PROGRAM INPUT_G6
VAR
	TMR11: TON;
	TMR12: TON;
	TMR10: TON;
	TMR8: TON;
	TMR9: TON;
	TMR7: TON;
	TMR3: TON;
	TP1: TP;
	TMR1: TON;
	START_ROBOT: TP;
	TP2: TP;
	O_G6_HANG: BOOL;
	I_G6_HANG: BOOL;
	TMR2: TON;
	GO_ROBOT: BOOL;
	TP3: TP;
	TMR4: TON;
	CNT_CYCLE: CTU;
	START_ROTATE: R_TRIG;
	IN: INT;
	TP_END_FUKUDA: TP;
	CNT_END_FUKUDA: CTU;
	ROBOT_READY: BOOL;
	ROBOT_G6_READY: BOOL;
	END_FUKUDA: BOOL;
	O_END_FUKUDA: BOOL;
	TEMP_COUNTER_FUKUDA_A: INT;
	TEMP_COUNTER_FUKUDA_B: INT;
	O_END_FUKUDB: BOOL;
	MAX_DEVICE: INT;
	TMR_HANG: TON;
	GRP1: Tp;
	GRP2: Tp;
	GRP3: Tp;
	GRP4: Tp;
	CNT_PLACING: ctu;
	CNT_TAKING: CTU;
	CNT_CYCLE1: CTU;
END_VAR

VAR PERSISTENT
	TRGEN: R_TRIG;
END_VAR

IF INPUT_G6_VAR.I_G6_ENABLE  THEN
//GRIPPING 
IF INPUT_G6_VAR.IX_G6_GRIPPER_1 THEN
	INPUT_G6_VAR.O_G6_GRIPPER_CLOSE_1:=TRUE;
	INPUT_G6_VAR.O_G6_GRIPPER_OPEN_1:=FALSE;
ELSE
	INPUT_G6_VAR.O_G6_GRIPPER_CLOSE_1:=FALSE;
	INPUT_G6_VAR.O_G6_GRIPPER_OPEN_1:=TRUE;
END_IF

IF INPUT_G6_VAR.IX_G6_GRIPPER_2 THEN
	INPUT_G6_VAR.O_G6_GRIPPER_CLOSE_2:=TRUE;
	INPUT_G6_VAR.O_G6_GRIPPER_OPEN_2:=FALSE;
ELSE
	INPUT_G6_VAR.O_G6_GRIPPER_CLOSE_2:=FALSE;
	INPUT_G6_VAR.O_G6_GRIPPER_OPEN_2:=TRUE;
END_IF 

IF INPUT_G6_VAR.IX_G6_GRIPPER_3 THEN
	INPUT_G6_VAR.O_G6_GRIPPER_CLOSE_3:=TRUE;
	INPUT_G6_VAR.O_G6_GRIPPER_OPEN_3:=FALSE;
ELSE
	INPUT_G6_VAR.O_G6_GRIPPER_CLOSE_3:=FALSE;
	INPUT_G6_VAR.O_G6_GRIPPER_OPEN_3:=TRUE;
END_IF

IF INPUT_G6_VAR.IX_G6_GRIPPER_4 THEN
	INPUT_G6_VAR.O_G6_GRIPPER_CLOSE_4:=TRUE;
	INPUT_G6_VAR.O_G6_GRIPPER_OPEN_4:=FALSE;
ELSE
	INPUT_G6_VAR.O_G6_GRIPPER_CLOSE_4:=FALSE;
	INPUT_G6_VAR.O_G6_GRIPPER_OPEN_4:=TRUE;
END_IF

//EXTENDER DOWN
IF INPUT_G6_VAR.IX_G6_GRIPPER_EXT_1 THEN
	INPUT_G6_VAR.O_G6_GRIPPER_EXT_DOWN_1:=TRUE;
	INPUT_G6_VAR.O_G6_GRIPPER_EXT_UP_1:=FALSE;
ELSE
	INPUT_G6_VAR.O_G6_GRIPPER_EXT_DOWN_1:=FALSE;
	INPUT_G6_VAR.O_G6_GRIPPER_EXT_UP_1:=TRUE;
END_IF

IF INPUT_G6_VAR.IX_G6_GRIPPER_EXT_2 THEN
	INPUT_G6_VAR.O_G6_GRIPPER_EXT_DOWN_2:=TRUE;
	INPUT_G6_VAR.O_G6_GRIPPER_EXT_UP_2:=FALSE;
ELSE
	INPUT_G6_VAR.O_G6_GRIPPER_EXT_DOWN_2:=FALSE;
	INPUT_G6_VAR.O_G6_GRIPPER_EXT_UP_2:=TRUE;
END_IF

IF INPUT_G6_VAR.IX_G6_GRIPPER_EXT_3 THEN
	INPUT_G6_VAR.O_G6_GRIPPER_EXT_DOWN_3:=TRUE;
	INPUT_G6_VAR.O_G6_GRIPPER_EXT_UP_3:=FALSE;
ELSE
	INPUT_G6_VAR.O_G6_GRIPPER_EXT_DOWN_3:=FALSE;
	INPUT_G6_VAR.O_G6_GRIPPER_EXT_UP_3:=TRUE;
END_IF

IF INPUT_G6_VAR.IX_G6_GRIPPER_EXT_4 THEN
	INPUT_G6_VAR.O_G6_GRIPPER_EXT_DOWN_4:=TRUE;
	INPUT_G6_VAR.O_G6_GRIPPER_EXT_UP_4:=FALSE;
ELSE
	INPUT_G6_VAR.O_G6_GRIPPER_EXT_DOWN_4:=FALSE;
	INPUT_G6_VAR.O_G6_GRIPPER_EXT_UP_4:=TRUE;
END_IF
IF INPUT_G6_VAR.I_G6_READY_TAKEUP THEN
	INPUT_G6_VAR.O_G6_GRIPPER_CLOSE_1:=FALSE;
	INPUT_G6_VAR.O_G6_GRIPPER_OPEN_1:=TRUE;
	
	INPUT_G6_VAR.O_G6_GRIPPER_CLOSE_2:=FALSE;
	INPUT_G6_VAR.O_G6_GRIPPER_OPEN_2:=TRUE;
	
	INPUT_G6_VAR.O_G6_GRIPPER_CLOSE_3:=FALSE;
	INPUT_G6_VAR.O_G6_GRIPPER_OPEN_3:=TRUE;
	
	INPUT_G6_VAR.O_G6_GRIPPER_CLOSE_3:=FALSE;
	INPUT_G6_VAR.O_G6_GRIPPER_OPEN_3:=TRUE;
END_IF

INPUT_G6_VAR.GRIPPER_OPEN_1:=INPUT_G6_VAR.I_G6_GRIPPER_OPEN_1;
INPUT_G6_VAR.GRIPPER_OPEN_2:=INPUT_G6_VAR.I_G6_GRIPPER_OPEN_2;
INPUT_G6_VAR.GRIPPER_OPEN_3:=INPUT_G6_VAR.I_G6_GRIPPER_OPEN_3;
INPUT_G6_VAR.GRIPPER_OPEN_4:=INPUT_G6_VAR.I_G6_GRIPPER_OPEN_4;

INPUT_G6_VAR.GRIPPER_CLOSE_1:=INPUT_G6_VAR.I_G6_GRIPPER_CLOSE_1;
INPUT_G6_VAR.GRIPPER_CLOSE_2:=INPUT_G6_VAR.I_G6_GRIPPER_CLOSE_2;
INPUT_G6_VAR.GRIPPER_CLOSE_3:=INPUT_G6_VAR.I_G6_GRIPPER_CLOSE_3;
INPUT_G6_VAR.GRIPPER_CLOSE_4:=INPUT_G6_VAR.I_G6_GRIPPER_CLOSE_4;

//ACTIVATE ROBOT
TRGEN(CLK:=INPUT_G6_VAR.I_G6_ENABLE); 
IF TRGEN.Q THEN
	INPUT_G6_VAR.O_G6_RESET_COUNTER_PICK:=TRUE;
END_IF
IF INPUT_G6_VAR.I_G6_START_PLACING OR INPUT_G6_VAR.I_G6_START_TAKEUP THEN
	INPUT_G6_VAR.O_G6_RESET_COUNTER_PICK:=FALSE;
END_IF
//IF INPUT_G6_VAR.I_G6_ENABLE THEN
TP_END_FUKUDA(IN:=INPUT_G6_VAR.I_G6_END_FUKUDA,PT:=T#0.1S);
CNT_END_FUKUDA(CU:=TP_END_FUKUDA.Q,RESET:=CNT_END_FUKUDA.Q,PV:=1000);

INPUT_VAR.I_STOPPER_TRANSFER_ON_A:= INPUT_VAR.O_STOPPER_TRANSFER_A;
//IF INPUT_VAR.I_STOPPER_TRANSFER_ON_A OR INPUT_VAR.I_STOPPER_TRANSFER_ON_B THEN
INPUT_G6_VAR.O_G6_SETMOTOROFF:=FALSE;
IF NOT INPUT_G6_VAR.I_G6_MOTORON THEN
	INPUT_G6_VAR.O_G6_STOP:=FALSE;
END_IF
IF NOT INPUT_G6_VAR.I_G6_MOTORON AND INPUT_G6_VAR.I_G6_READY AND NOT INPUT_G6_VAR.I_G6_ESTOPON AND NOT INPUT_G6_VAR.I_G6_SAFEGUARDON THEN
	INPUT_G6_VAR.O_G6_SETMOTORON:=TRUE;
	INPUT_G6_VAR.O_G6_STOP:=FALSE;
	INPUT_G6_VAR.O_G6_RESET :=FALSE;	
	INPUT_G6_VAR.O_G6_START :=FALSE ;
	INPUT_G6_VAR.O_G6_CONTINUE :=FALSE;
TMR1(IN:=INPUT_G6_VAR.O_G6_SETMOTORON ,PT:=T#0.5S);
ELSE
	INPUT_G6_VAR.O_G6_SETMOTOROFF:=FALSE;
	INPUT_G6_VAR.O_G6_SETMOTORON:=FALSE;
END_IF

//START POSITION CANNOT BE 0
IF INPUT_G6_VAR.START_POSITION =0 THEN
	INPUT_G6_VAR.START_POSITION :=1;
END_IF
// ERROR OVERRIDE	
	IF 	INPUT_G6_VAR.I_G6_ERROR OR INPUT_G6_VAR.I_CMDERROR THEN// AND INPUT_G6_VAR.I_G6_READY THEN// OR INPUT_G6_VAR.G6_ERROR1> 0 OR INPUT_G6_VAR.G6_ERROR2 > 0 THEN
		INPUT_G6_VAR.O_G6_STOP :=TRUE ;			
		TMR10(IN:=INPUT_G6_VAR.O_G6_STOP,PT:=T#1S);
		INPUT_VAR.ALARM1:=INPUT_G6_VAR.I_G6_ERROR OR INPUT_G6_VAR.G6_ERROR1> 0 OR INPUT_G6_VAR.G6_ERROR2 > 0;
		IF NOT TMR10.Q AND INPUT_G6_VAR.I_G6_READY THEN
			INPUT_G6_VAR.O_G6_RESET :=TRUE;	
			INPUT_G6_VAR.O_G6_START :=FALSE ;
			INPUT_G6_VAR.O_G6_CONTINUE :=FALSE;
			INPUT_G6_VAR.O_G6_STOP :=FALSE ;	
			TMR10(IN:=FALSE);
		END_IF
	ELSE
		INPUT_G6_VAR.O_G6_RESET :=FALSE;	
	END_IF
IF INPUT_G6_VAR.I_G6_MOTORON AND NOT INPUT_G6_VAR.I_G6_ESTOPON AND NOT INPUT_G6_VAR.I_G6_SAFEGUARDON AND INDEXING_1_VAR.I_INDEXING_1_ROTATION_DONE  THEN
IF (INPUT_G6_VAR.I_G6_READY OR INPUT_G6_VAR.I_G6_RUNNING) AND NOT INPUT_G6_VAR.I_G6_ERROR AND NOT INPUT_G6_VAR.I_CMDERROR THEN
	
//START FOR 1ST TIME
		IF INPUT_G6_VAR.I_G6_READY  AND NOT INPUT_G6_VAR.I_G6_RUNNING THEN
			INPUT_G6_VAR.O_G6_STOP:=FALSE;
			INPUT_G6_VAR.O_G6_CONTINUE :=FALSE;
			INPUT_G6_VAR.O_G6_PAUSE:=FALSE;
			INPUT_G6_VAR.O_G6_RESET :=FALSE;
			TMR7(IN:=INPUT_G6_VAR.I_G6_READY,PT:=T#1S);
			START_ROBOT(IN:=TMR7.Q,PT:=T#2S);
			INPUT_G6_VAR.O_G6_START :=TMR7.Q ;
		ELSE
			TMR7(IN:=FALSE);
			INPUT_G6_VAR.O_G6_START :=FALSE ;
		END_IF
		IF  NOT INPUT_G6_VAR.I_G6_READY OR INPUT_G6_VAR.I_G6_RUNNING THEN
			INPUT_G6_VAR.O_G6_START :=FALSE ;
		END_IF
		IF INPUT_G6_VAR.I_G6_READY AND INPUT_G6_VAR.O_G6_START THEN
			TMR_HANG(IN:=TRUE,PT:=T#30S);
			IF TMR_HANG.Q THEN
				INPUT_G6_VAR.O_G6_START :=FALSE ;
				INPUT_G6_VAR.O_G6_STOP :=TRUE ;
			END_IF
		ELSE
			TMR_HANG(IN:=FALSE);
		END_IF
//STOP 
		IF INPUT_G6_VAR.I_G6_END_FUKUDA OR( NOT INPUT_G6_VAR.I_G6_READY AND NOT INPUT_G6_VAR.I_G6_RUNNING) THEN
			TMR8(IN:=FALSE);
			TMR9(IN:=FALSE);
		//	INPUT_G6_VAR.O_G6_STOP:=TRUE;
		//	LOADER_RS4_VAR.O_LOADER_RS4_STOP:=TRUE;
		END_IF
		TMR2(IN:=INPUT_G6_VAR.O_G6_STOP,PT:=T#1S);
		IF TMR2.Q THEN
			INPUT_G6_VAR.I_G6_HANG:=FALSE;
			INPUT_G6_VAR.O_G6_STOP:=FALSE;
			TMR1(IN:=FALSE);
		END_IF

		
//CONTINUE	
		//INPUT_G6_VAR.GO_ROBOT:=(INPUT_G6_VAR.I_G6_READY_PLACING AND LOADER_RS4_VAR.I_LOADER_RS4_READY_TAKEUP AND INDEXING_2_VAR.O_ROTATION_DONE )OR(INPUT_G6_VAR.I_G6_READY_PLACING AND NOT LOADER_RS4_VAR.I_LOADER_RS4_ENABLE AND  INDEXING_1_VAR.I_INDEXING_1_ROTATION_DONE)    ;	
		IF (INPUT_G6_VAR.I_G6_READY_PLACING AND LOADER_RS4_VAR.I_LOADER_RS4_READY_TAKEUP AND  INDEXING_1_VAR.I_INDEXING_1_ROTATION_DONE AND INDEXING_2_VAR.I_INDEXING_2_ROTATION_DONE)  THEN
			INPUT_G6_VAR.GO_ROBOT:=TRUE;
		END_IF
		IF (INPUT_G6_VAR.I_G6_READY_PLACING AND NOT LOADER_RS4_VAR.I_LOADER_RS4_ENABLE AND  INDEXING_1_VAR.I_INDEXING_1_ROTATION_DONE AND INDEXING_2_VAR.I_INDEXING_2_ROTATION_DONE) THEN
			INPUT_G6_VAR.GO_ROBOT:=TRUE;
		END_IF
		IF INPUT_G6_VAR.I_G6_START_TAKEUP THEN
			INPUT_G6_VAR.GO_ROBOT:=FALSE;
		END_IF	
		IF INDEXING_1_VAR.I_INDEXING_1_ROTATION_DONE AND INPUT_G6_VAR.GO_ROBOT AND INPUT_VAR.STRAIGHTEN_DONE  AND INPUT_G6_VAR.I_G6_RUNNING AND NOT LOADER_RS4_VAR.I_LOADER_RS4_END_CARRIER THEN
			TMR3(IN:=INPUT_G6_VAR.GO_ROBOT ,PT:=T#0.5S);
			TP1(IN:=INPUT_G6_VAR.GO_ROBOT,PT:=T#0.1S);
		ELSE
			TMR3(IN:=FALSE);
			TP1(IN:=FALSE);
		END_IF
		
		IF INPUT_G6_VAR.I_G6_RUNNING AND  INDEXING_1_VAR.I_INDEXING_1_ROTATION_DONE THEN
			INPUT_G6_VAR.O_G6_START :=FALSE ;
			INPUT_G6_VAR.O_G6_CONTINUE :=TMR3.Q;
			IF (CNT_CYCLE.CV <=3 AND INPUT_G6_VAR.I_G6_READY_TAKEUP AND (INPUT_VAR.I_FUKUDA_TRANSFER_AT_FRONT_A OR INPUT_VAR.I_FUKUDA_TRANSFER_AT_FRONT_B)) AND  INDEXING_1_VAR.I_INDEXING_1_ROTATION_DONE THEN
				INPUT_G6_VAR.O_G6_CONTINUE :=TRUE;
			END_IF
		END_IF
		
//ENABLE ROBOT LOADER RS4
		CNT_CYCLE(CU:=INPUT_G6_VAR.I_G6_START_PLACING,RESET:=NOT INPUT_G6_VAR.I_G6_ENABLE,PV:=4);
		IF CNT_CYCLE.CV =3 AND NOT LOADER_RS4_VAR.I_LOADER_RS4_ENABLE  THEN
			LOADER_RS4_VAR.I_LOADER_RS4_ENABLE:=TRUE;
		END_IF
//PAUSE
		CNT_CYCLE1(CU:=INPUT_G6_VAR.I_G6_START_TAKEUP,RESET:=NOT INPUT_G6_VAR.I_G6_ENABLE,PV:=5);
		IF CNT_CYCLE.CV >=4 AND NOT LOADER_RS4_VAR.I_LOADER_RS4_ENABLE AND  INPUT_G6_VAR.I_G6_RUNNING THEN
			///INPUT_G6_VAR.O_G6_PAUSE:=TRUE;
		END_IF
//START ROTATE INDEXING 1
		IF NOT LOADER_RS4_VAR.I_LOADER_RS4_ENABLE  AND  (INPUT_G6_VAR.IX_G6_GRIPPER_EXT_1 AND INPUT_G6_VAR.I_G6_START_TAKEUP )  THEN
			START_ROTATE(CLK:=TRUE);
			INDEXING_1_VAR.O_ROTATION_START:=TRUE;
		ELSE
			START_ROTATE(CLK:=FALSE);
		END_IF
		IF INPUT_G6_VAR.I_G6_START_PLACING THEN
			INDEXING_1_VAR.O_ROTATION_START:=FALSE;
		END_IF
		
 //SYNCRONIZE ROBOT G6 AND RS4 
		IF INPUT_G6_VAR.I_G6_START_TAKEUP AND LOADER_RS4_VAR.I_LOADER_RS4_START_PLACING  THEN
			INPUT_G6_VAR.GO_ROBOT:=FALSE;
			INPUT_G6_VAR.I_READY_CONTINUE:=FALSE;
			LOADER_RS4_VAR.I_READY_CONTINUE:=FALSE;
		END_IF
		
		IF INPUT_G6_VAR.I_READY_CONTINUE AND LOADER_RS4_VAR.I_READY_CONTINUE THEN
			//INPUT_G6_VAR.O_G6_CONTINUE :=TRUE;
			//LOADER_RS4_VAR.O_LOADER_RS4_CONTINUE :=TRUE;
		END_IF
		
 //END FUKUDA21
 //INPUT_G6_VAR.I_MAX_DEVICE:=40;
// IF INPUT_G6_VAR.I_G6_START_takeup THEN
	 TEMP_COUNTER_FUKUDA_A:=INPUT_G6_VAR.COUNTER_FUKUDA_A;
	 TEMP_COUNTER_FUKUDA_B:=INPUT_G6_VAR.COUNTER_FUKUDA_B;
// END_IF
 		
		IF TEMP_COUNTER_FUKUDA_A >=INPUT_G6_VAR.I_MAX_DEVICE   OR TEMP_COUNTER_FUKUDA_B >=INPUT_G6_VAR.I_MAX_DEVICE THEN
			INPUT_G6_VAR.O_G6_RESET_COUNTER_PICK:=TRUE;
			INPUT_G6_VAR.START_POSITION:=1;
			//TEMP_COUNTER_FUKUDA_A:=0;
			ELSE
				INPUT_G6_VAR.O_G6_RESET_COUNTER_PICK:=FALSE;
		END_IF
		
		IF TEMP_COUNTER_FUKUDA_A >=INPUT_G6_VAR.I_MAX_DEVICE THEN
			O_END_FUKUDA:=TRUE;
			//INPUT_G6_VAR.O_G6_SELECT_FUKUDA_A:=TRUE;
			//INPUT_VAR.I_FUKUDA_TRANSFER_A_PICK_DONE:=TRUE;
			//TEMP_COUNTER_FUKUDA_A:=0;
			ELSE
				O_END_FUKUDA:=FALSE;
		END_IF
		
		IF TEMP_COUNTER_FUKUDA_B >=INPUT_G6_VAR.I_MAX_DEVICE THEN
			O_END_FUKUDB:=TRUE;
			//INPUT_G6_VAR.O_G6_SELECT_FUKUDA_A:=FALSE;
			//INPUT_VAR.I_FUKUDA_TRANSFER_B_PICK_DONE:=TRUE;
			ELSE
			O_END_FUKUDB:=FALSE;
		END_IF

	IF INPUT_G6_VAR.O_G6_GRIPPER_CLOSE_1  THEN
 		GRP1(IN:=TRUE,PT:=T#0.1S);
		ELSE
		GRP1(IN:=FALSE);	
	END_IF
	IF INPUT_G6_VAR.O_G6_GRIPPER_CLOSE_2  THEN
 		GRP2(IN:=TRUE,PT:=T#0.1S); 
		ELSE
		GRP2(IN:=FALSE);	
	END_IF
	IF INPUT_G6_VAR.O_G6_GRIPPER_CLOSE_3  THEN
 		GRP3(IN:=TRUE,PT:=T#0.1S);
		ELSE
		GRP3(IN:=FALSE);	
	END_IF
	IF INPUT_G6_VAR.O_G6_GRIPPER_CLOSE_4  THEN
 		GRP4(IN:=TRUE,PT:=T#0.1S);
		ELSE
		GRP4(IN:=FALSE);	
	END_IF
//	IF LOADER_RS4_VAR.I_LOADER_RS4_START_PLACING THEN
		CNT_TAKING.CU:=(GRP1.Q OR GRP2.Q OR GRP3.Q OR GRP4.Q); 
//	END_IF
	CNT_PLACING(RESET:=INDEXING_2_VAR.O_ROTATION_START,PV:=68);

END_IF
END_IF
ELSE
	//INPUT_G6_VAR.O_G6_STOP :=TRUE ;
	//INPUT_G6_VAR.O_G6_RESET :=TRUE;	
	(*INPUT_G6_VAR.O_G6_START :=FALSE ;
	INPUT_G6_VAR.O_G6_CONTINUE :=FALSE;
	
	INPUT_G6_VAR.O_G6_SETMOTORON:=FALSE;
	
	INPUT_G6_VAR.O_G6_GRIPPER_EXT_DOWN_1:=FALSE;
	INPUT_G6_VAR.O_G6_GRIPPER_EXT_UP_1:=TRUE;
	
	INPUT_G6_VAR.O_G6_GRIPPER_EXT_DOWN_2:=FALSE;
	INPUT_G6_VAR.O_G6_GRIPPER_EXT_UP_2:=TRUE;
	
	INPUT_G6_VAR.O_G6_GRIPPER_EXT_DOWN_3:=FALSE;
	INPUT_G6_VAR.O_G6_GRIPPER_EXT_UP_3:=TRUE;
	
	INPUT_G6_VAR.O_G6_GRIPPER_EXT_DOWN_4:=FALSE;
	INPUT_G6_VAR.O_G6_GRIPPER_EXT_UP_4:=TRUE;
	
	IF INPUT_G6_VAR.I_G6_READY THEN
		INPUT_G6_VAR.O_G6_SETMOTOROFF:=TRUE;
	END_IF
	*)
END_IF
//END_IF

END_PROGRAM

(* stored: Version 1.1.0.1, ProductVersion 3.1.4020.12
   POU INPUT_G6: Id {90f5e18c-05ba-44d3-9e34-0b58d9ccefe9}, SpecialFunc None *)
